FUNCTION fSetCylinderVelocity : REAL
VAR_INPUT
END_VAR
VAR
END_VAR

END_FUNCTION

(* stored: Version 1.1.0.1, ProductVersion 3.1.4024.10
   POU fSetCylinderVelocity: Id {d9ceb50e-9842-4b82-bfea-7606e70d0f60}, SpecialFunc None *)
